% RSLogix 500 project PROJECT5-DIGITALROTAMETER.RSS, saved by version 8.30.00.16 %
PROJECT "UNTITLED"    % processor: Bul.1763 MicroLogix 1100 Series B %

PROGRAM FILES
  LAD 2   6 rungs

DATA FILES
  O0 OUTPUT  4 elements
  I1 INPUT  6 elements
  S2 STATUS  66 elements
  B3 BINARY  1 elements
  T4 TIMER  2 elements
  C5 COUNTER  1 elements
  R6 CONTROL  1 elements
  N7 INTEGER  1 elements
  F8 FLOAT  3 elements

LADDER 2
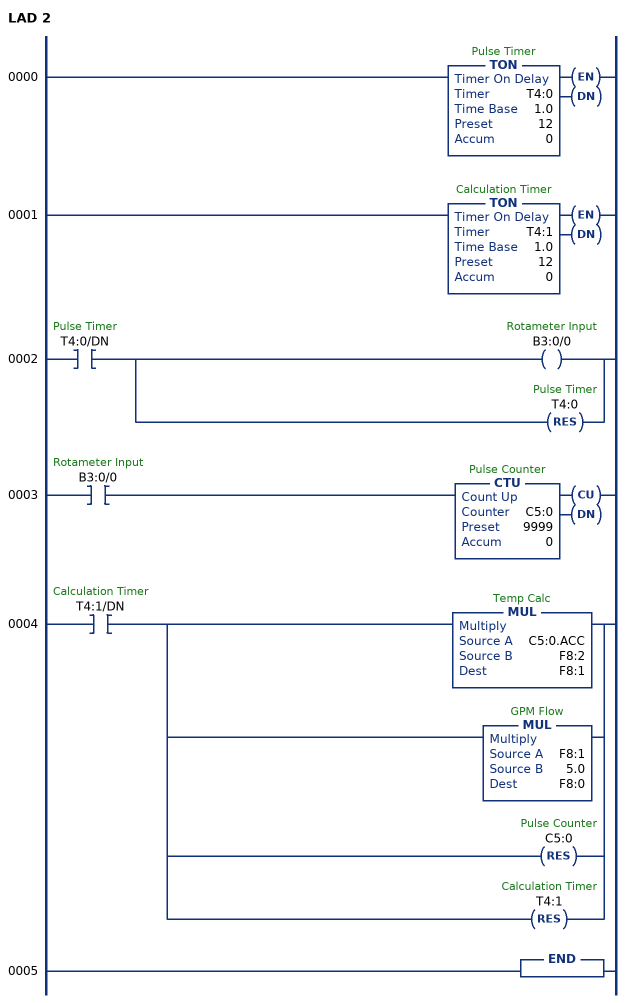
% Rung: 0 %
SOR TON T4:0 1.0 12 0 EOR
%   T4:0  "Pulse Timer" %
% Rung: 1 %
SOR TON T4:1 1.0 12 0 EOR
%   T4:1  "Calculation Timer" %
% Rung: 2 %
SOR XIC T4:0/DN BST OTE B3:0/0 NXB RES T4:0 BND EOR
%   T4:0  "Pulse Timer" %
%   B3:0/0  "Rotameter Input" %
% Rung: 3 %
SOR XIC B3:0/0 CTU C5:0 9999 0 EOR
%   B3:0/0  "Rotameter Input" %
%   C5:0  "Pulse Counter" %
% Rung: 4 %
SOR XIC T4:1/DN BST MUL C5:0.ACC F8:2 F8:1 NXB MUL F8:1 5.0 F8:0 NXB RES C5:0 NXB RES T4:1 BND EOR
%   T4:1  "Calculation Timer" %
%   C5:0  "Pulse Counter" %
%   F8:2  "Oil per pulse (Gallons)" %
%   F8:1  "Temp Calc" %
%   F8:0  "GPM Flow" %
% Rung: 5 %
SOR END EOR

DATA TABLE (non-zero values as saved)
DATA T4
% .PRE .ACC %
% T4:0 % 12 0
% T4:1 % 12 0
DATA C5
% .PRE .ACC %
% C5:0 % 9999 0
DATA F8
% F8:0 % 189 37.8 6.3
